// SIMATIC S7-200 project (STEP 7-Micro/WIN), CPU 226 CN REL 02.01

ORGANIZATION_BLOCK MAIN:OB1
TITLE=程序注释
BEGIN
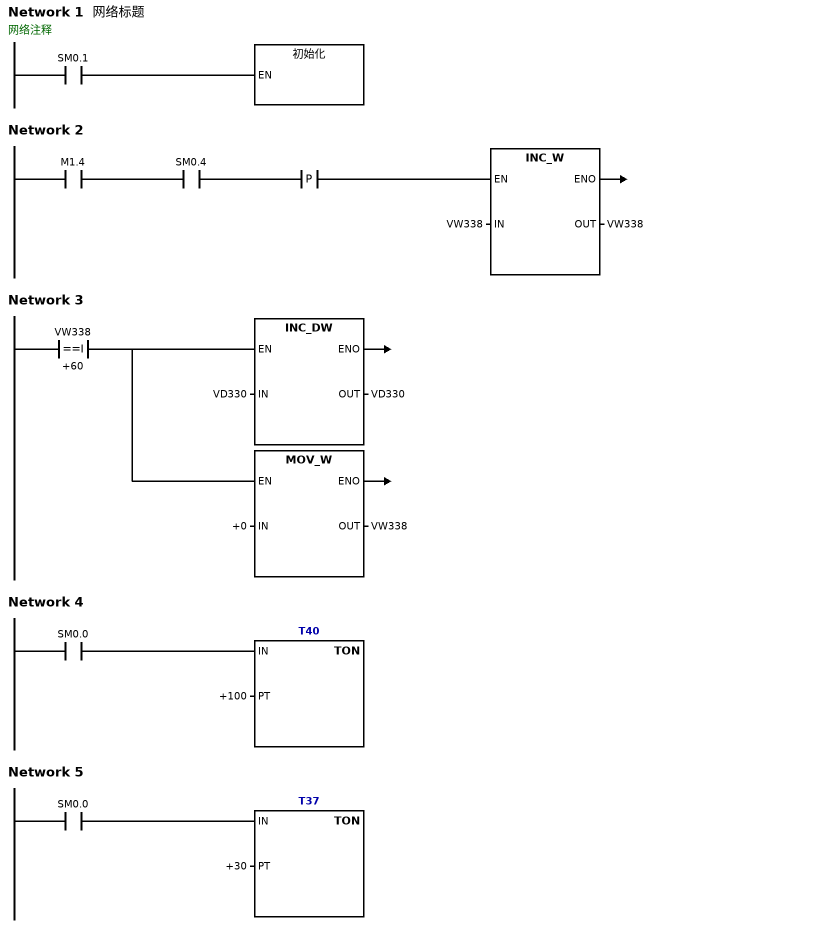
Network 1 // 网络标题
// 网络注释
LD     SM0.1
CALL   初始化:SBR0
Network 2
LD     M1.4
A      SM0.4
EU
INCW   VW338
Network 3
LDW=   VW338, +60
INCD   VD330
MOVW   +0, VW338
Network 4
LD     SM0.0
TON    T40, +100
Network 5
LD     SM0.0
TON    T37, +30
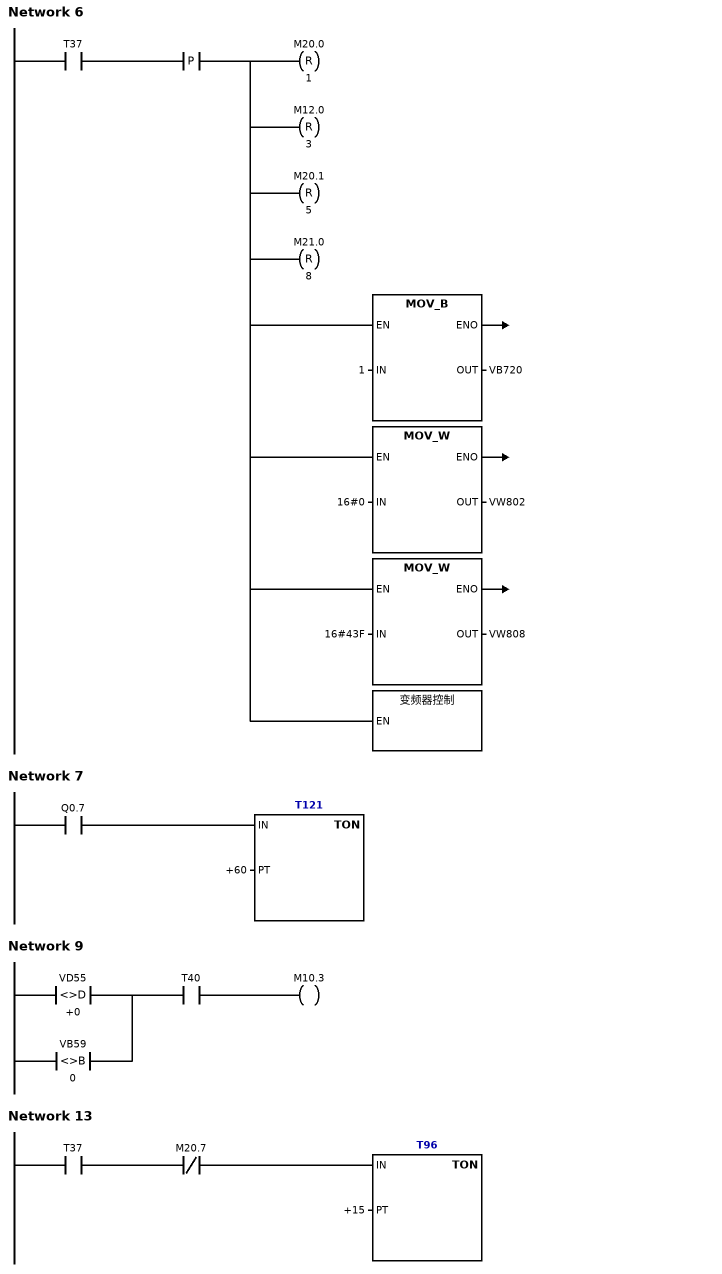
Network 6
LD     T37
EU
R      M20.0, 1
R      M12.0, 3
R      M20.1, 5
R      M21.0, 8
MOVB   1, VB720
MOVW   16#0, VW802
MOVW   16#43F, VW808
CALL   变频器控制:SBR16
Network 7
LD     Q0.7
TON    T121, +60
Network 9
LDD<>  VD55, +0
OB<>   VB59, 0
A      T40
=      M10.3
Network 13
LD     T37
AN     M20.7
TON    T96, +15
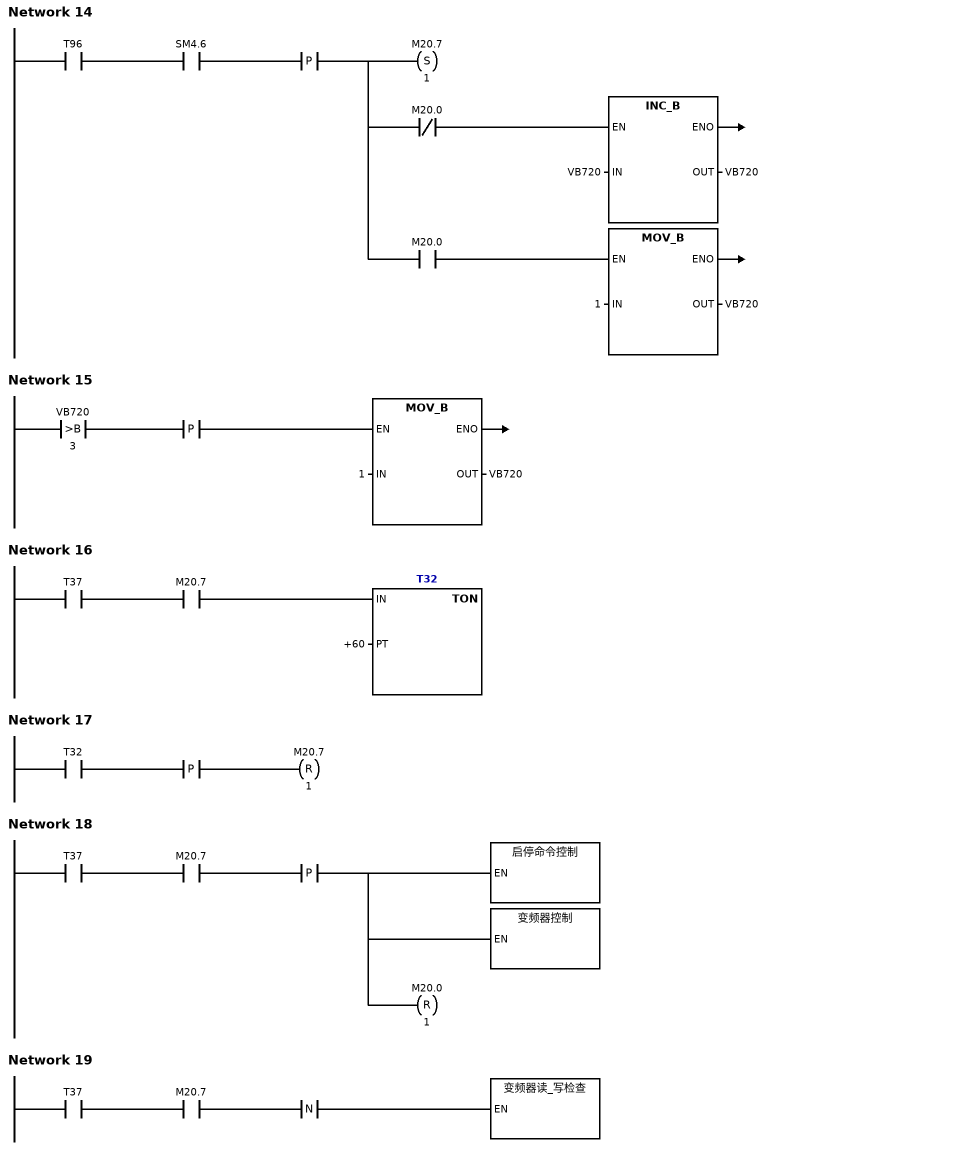
Network 14
LD     T96
A      SM4.6
EU
LPS
S      M20.7, 1
AN     M20.0
INCB   VB720
LPP
A      M20.0
MOVB   1, VB720
Network 15
LDB>   VB720, 3
EU
MOVB   1, VB720
Network 16
LD     T37
A      M20.7
TON    T32, +60
Network 17
LD     T32
EU
R      M20.7, 1
Network 18
LD     T37
A      M20.7
EU
CALL   启停命令控制:SBR4
CALL   变频器控制:SBR16
R      M20.0, 1
Network 19
LD     T37
A      M20.7
ED
CALL   变频器读_写检查:SBR3
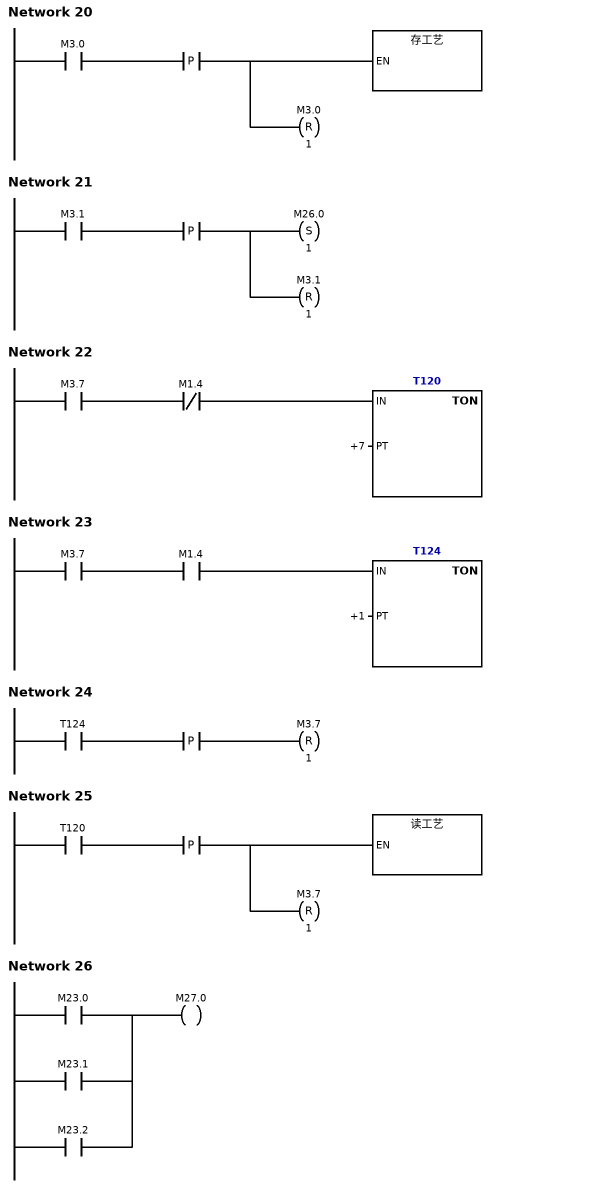
Network 20
LD     M3.0
EU
CALL   存工艺:SBR5
R      M3.0, 1
Network 21
LD     M3.1
EU
S      M26.0, 1
R      M3.1, 1
Network 22
LD     M3.7
AN     M1.4
TON    T120, +7
Network 23
LD     M3.7
A      M1.4
TON    T124, +1
Network 24
LD     T124
EU
R      M3.7, 1
Network 25
LD     T120
EU
CALL   读工艺:SBR6
R      M3.7, 1
Network 26
LD     M23.0
O      M23.1
O      M23.2
=      M27.0
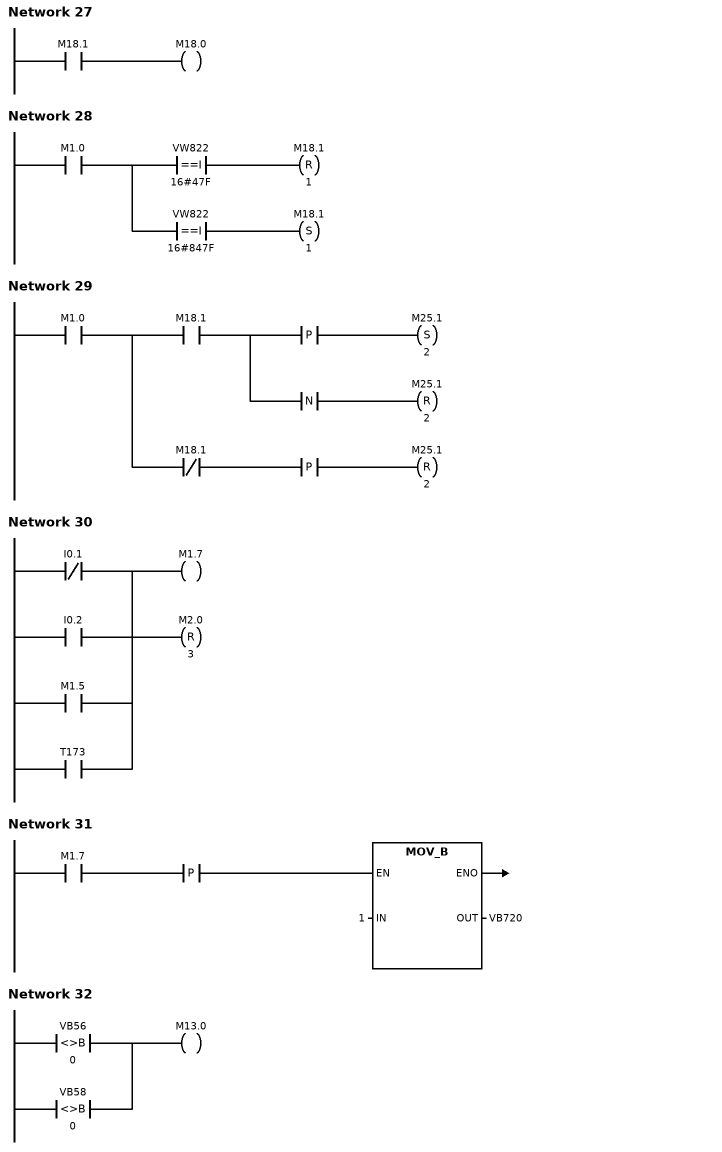
Network 27
LD     M18.1
=      M18.0
Network 28
LD     M1.0
LPS
AW=    VW822, 16#47F
R      M18.1, 1
LPP
AW=    VW822, 16#847F
S      M18.1, 1
Network 29
LD     M1.0
LPS
A      M18.1
LPS
EU
S      M25.1, 2
LPP
ED
R      M25.1, 2
LPP
AN     M18.1
EU
R      M25.1, 2
Network 30
LDN    I0.1
O      I0.2
O      M1.5
O      T173
=      M1.7
R      M2.0, 3
Network 31
LD     M1.7
EU
MOVB   1, VB720
Network 32
LDB<>  VB56, 0
OB<>   VB58, 0
=      M13.0
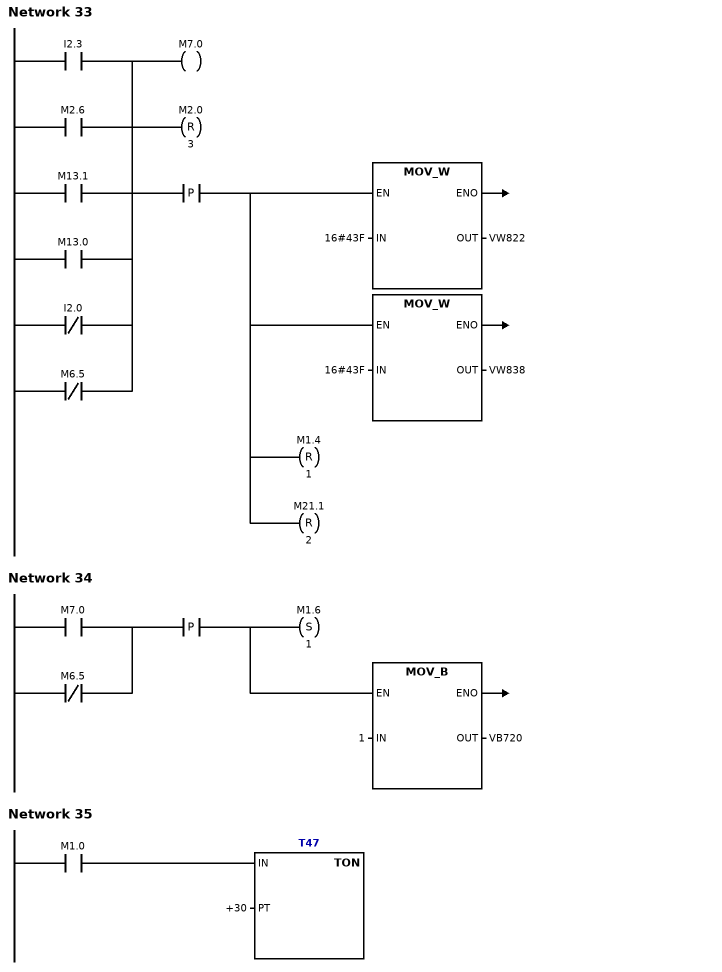
Network 33
LD     I2.3
O      M2.6
O      M13.1
O      M13.0
ON     I2.0
ON     M6.5
=      M7.0
R      M2.0, 3
EU
MOVW   16#43F, VW822
MOVW   16#43F, VW838
R      M1.4, 1
R      M21.1, 2
Network 34
LD     M7.0
ON     M6.5
EU
S      M1.6, 1
MOVB   1, VB720
Network 35
LD     M1.0
TON    T47, +30
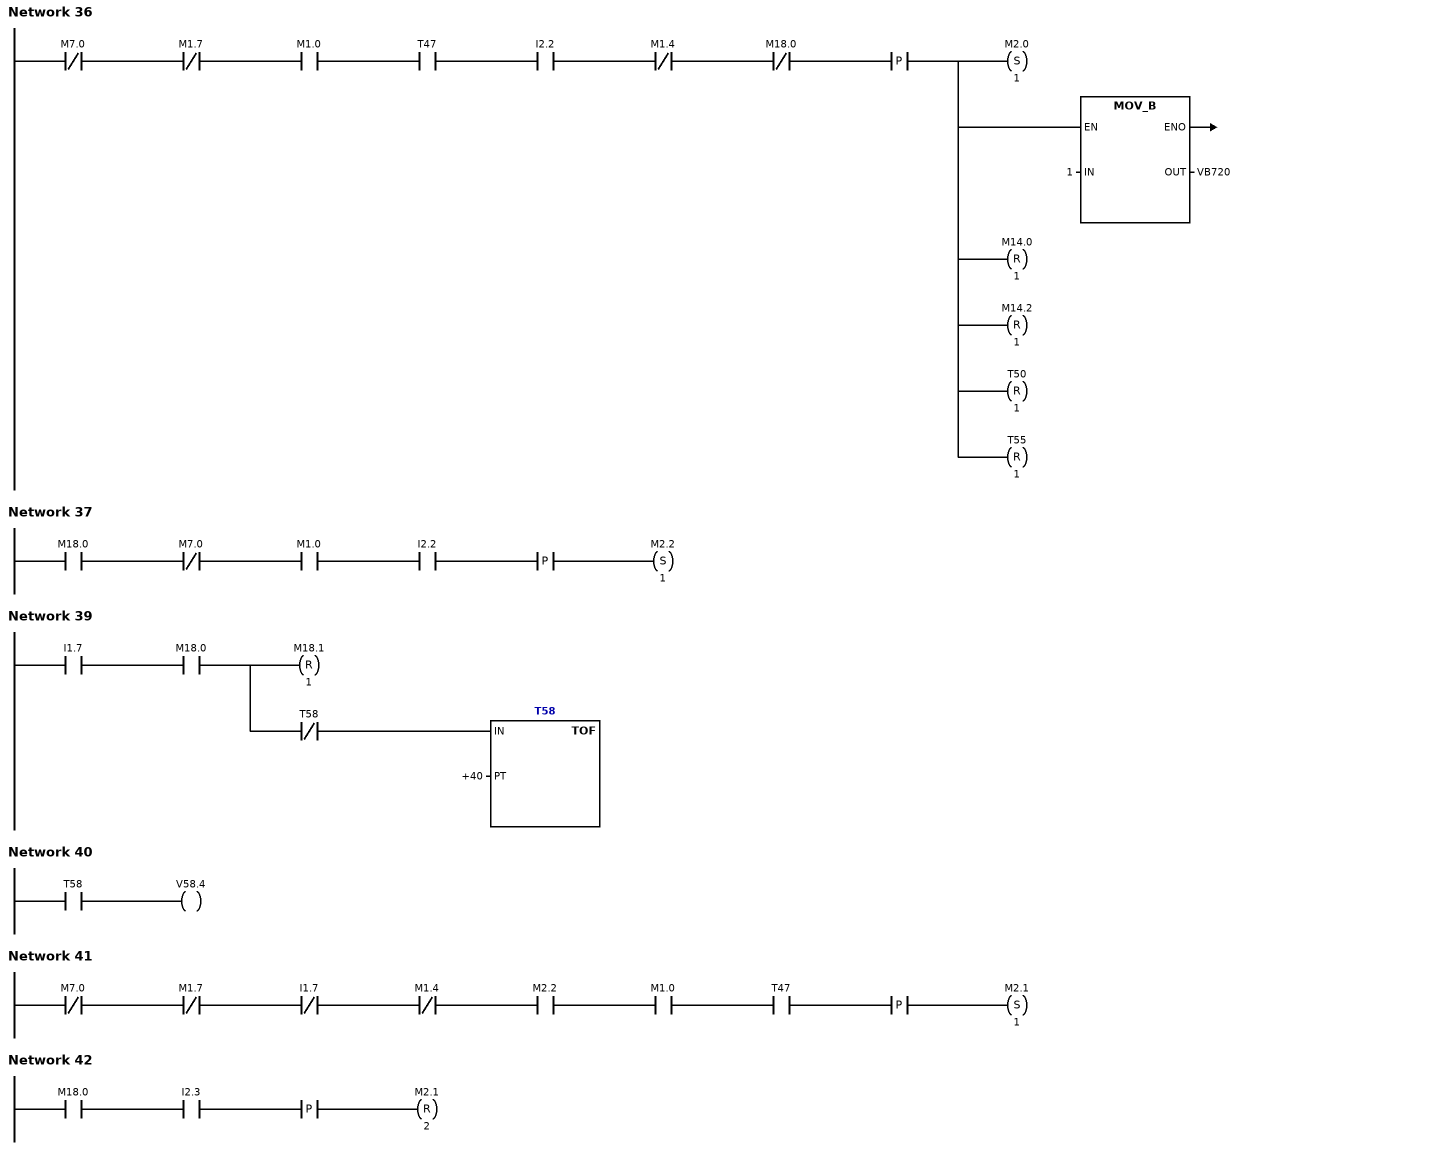
Network 36
LDN    M7.0
AN     M1.7
A      M1.0
A      T47
A      I2.2
AN     M1.4
AN     M18.0
EU
S      M2.0, 1
MOVB   1, VB720
R      M14.0, 1
R      M14.2, 1
R      T50, 1
R      T55, 1
Network 37
LD     M18.0
AN     M7.0
A      M1.0
A      I2.2
EU
S      M2.2, 1
Network 39
LD     I1.7
A      M18.0
R      M18.1, 1
AN     T58
TOF    T58, +40
Network 40
LD     T58
=      V58.4
Network 41
LDN    M7.0
AN     M1.7
AN     I1.7
AN     M1.4
A      M2.2
A      M1.0
A      T47
EU
S      M2.1, 1
Network 42
LD     M18.0
A      I2.3
EU
R      M2.1, 2
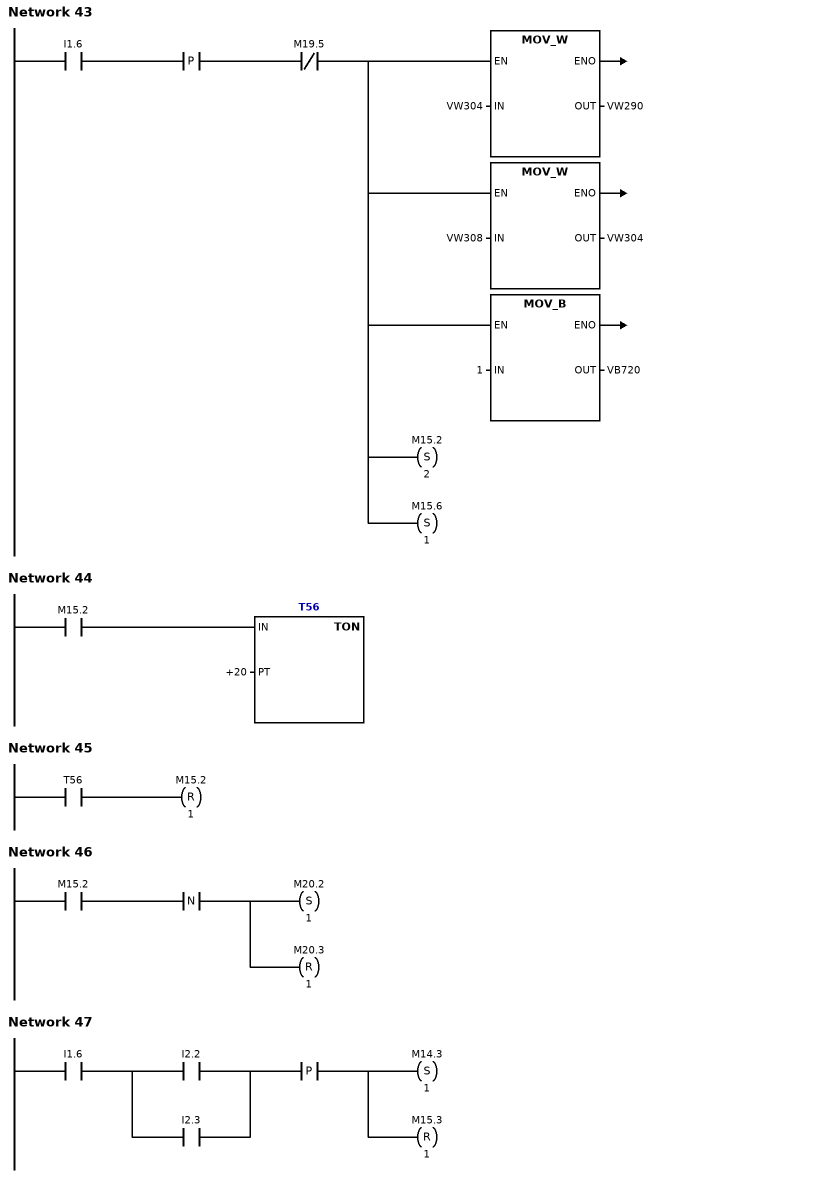
Network 43
LD     I1.6
EU
AN     M19.5
MOVW   VW304, VW290
MOVW   VW308, VW304
MOVB   1, VB720
S      M15.2, 2
S      M15.6, 1
Network 44
LD     M15.2
TON    T56, +20
Network 45
LD     T56
R      M15.2, 1
Network 46
LD     M15.2
ED
S      M20.2, 1
R      M20.3, 1
Network 47
LD     I1.6
LD     I2.2
O      I2.3
ALD
EU
S      M14.3, 1
R      M15.3, 1
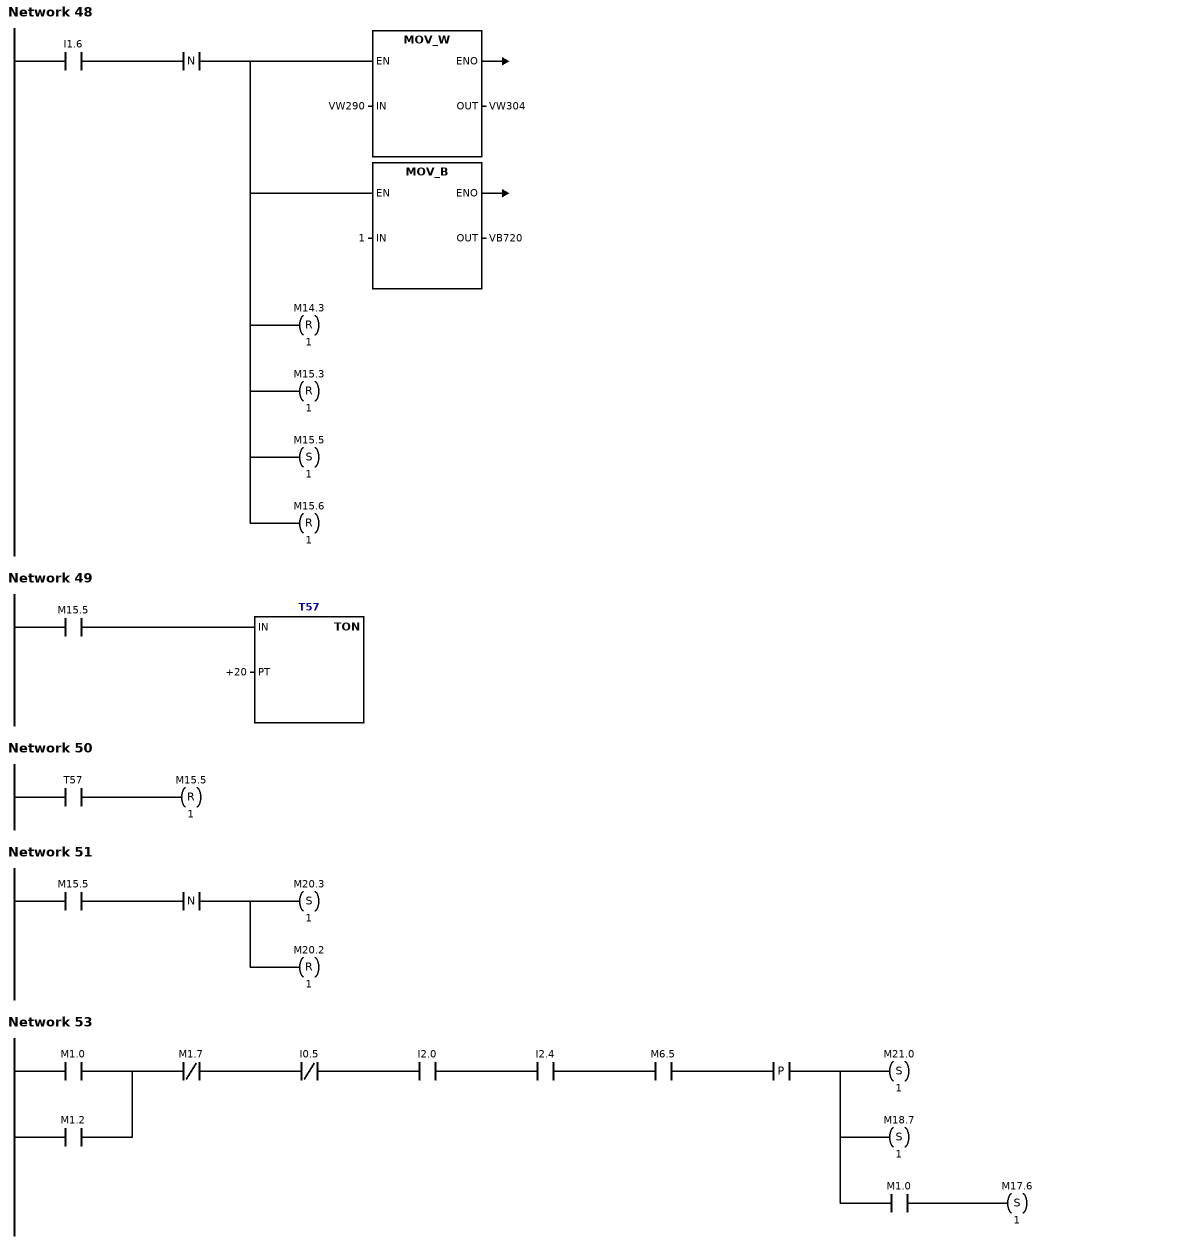
Network 48
LD     I1.6
ED
MOVW   VW290, VW304
MOVB   1, VB720
R      M14.3, 1
R      M15.3, 1
S      M15.5, 1
R      M15.6, 1
Network 49
LD     M15.5
TON    T57, +20
Network 50
LD     T57
R      M15.5, 1
Network 51
LD     M15.5
ED
S      M20.3, 1
R      M20.2, 1
Network 53
LD     M1.0
O      M1.2
AN     M1.7
AN     I0.5
A      I2.0
A      I2.4
A      M6.5
EU
S      M21.0, 1
S      M18.7, 1
A      M1.0
S      M17.6, 1
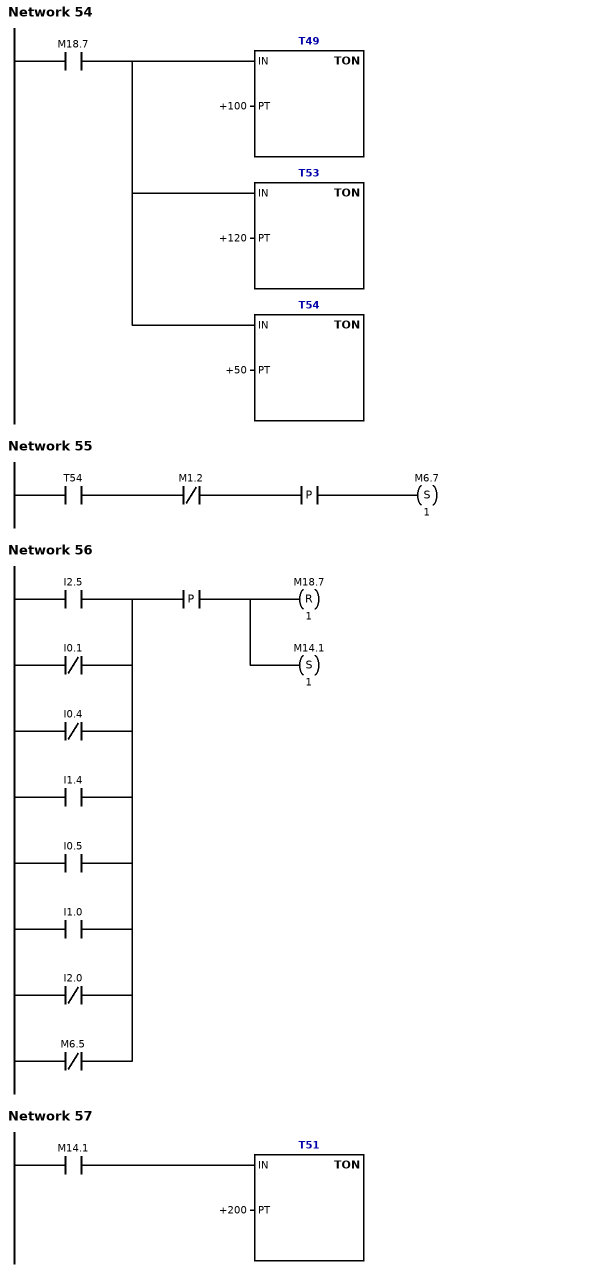
Network 54
LD     M18.7
TON    T49, +100
TON    T53, +120
TON    T54, +50
Network 55
LD     T54
AN     M1.2
EU
S      M6.7, 1
Network 56
LD     I2.5
ON     I0.1
ON     I0.4
O      I1.4
O      I0.5
O      I1.0
ON     I2.0
ON     M6.5
EU
R      M18.7, 1
S      M14.1, 1
Network 57
LD     M14.1
TON    T51, +200
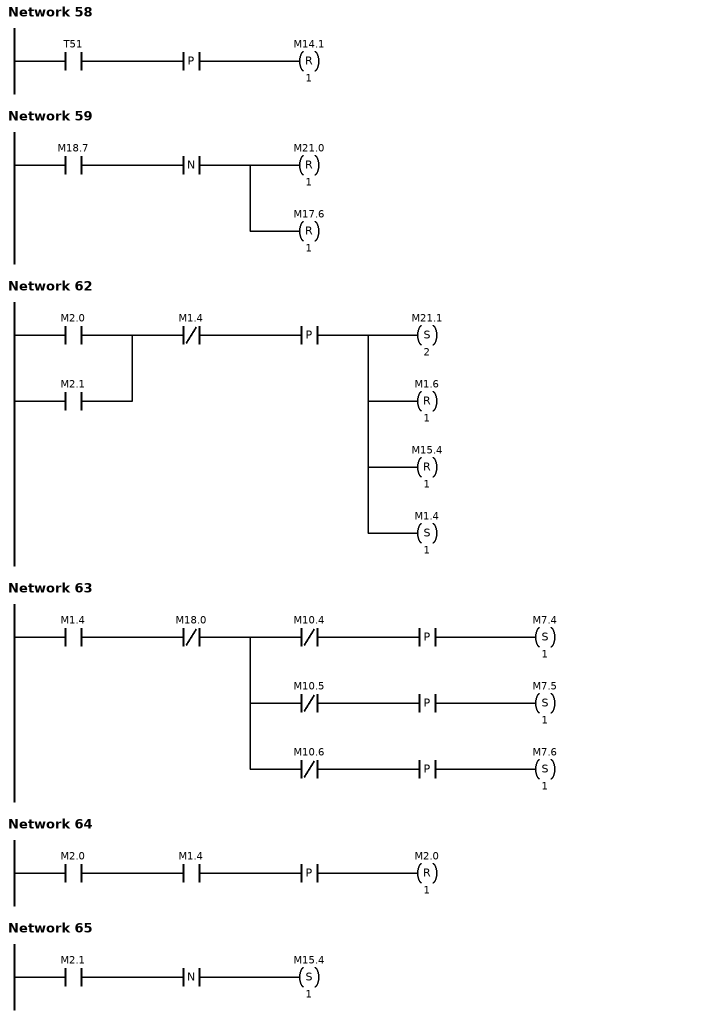
Network 58
LD     T51
EU
R      M14.1, 1
Network 59
LD     M18.7
ED
R      M21.0, 1
R      M17.6, 1
Network 62
LD     M2.0
O      M2.1
AN     M1.4
EU
S      M21.1, 2
R      M1.6, 1
R      M15.4, 1
S      M1.4, 1
Network 63
LD     M1.4
AN     M18.0
LPS
AN     M10.4
EU
S      M7.4, 1
LRD
AN     M10.5
EU
S      M7.5, 1
LPP
AN     M10.6
EU
S      M7.6, 1
Network 64
LD     M2.0
A      M1.4
EU
R      M2.0, 1
Network 65
LD     M2.1
ED
S      M15.4, 1
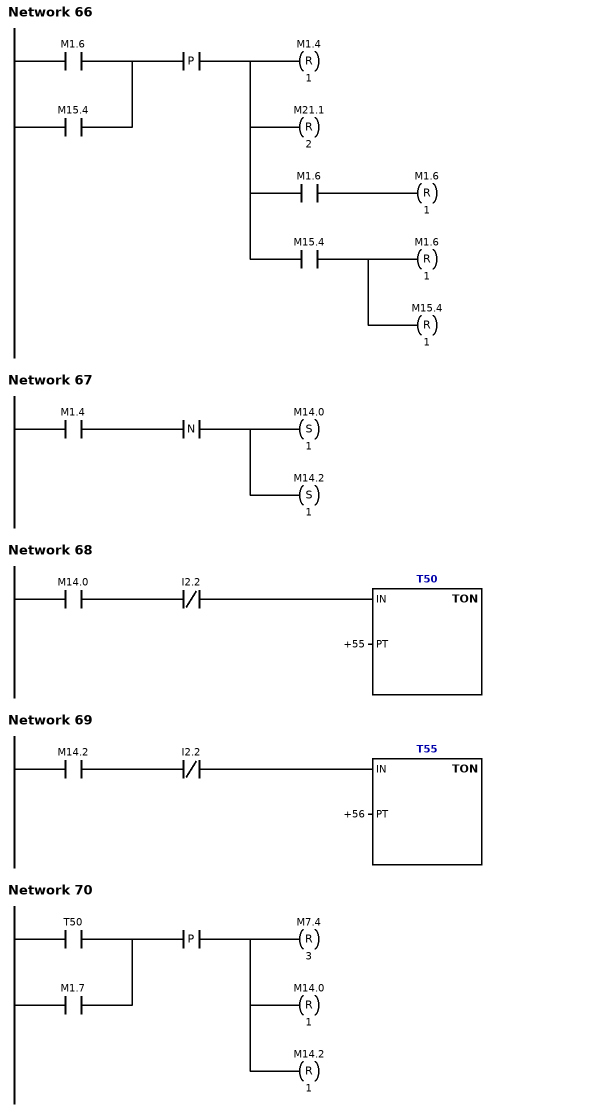
Network 66
LD     M1.6
O      M15.4
EU
LPS
R      M1.4, 1
R      M21.1, 2
A      M1.6
R      M1.6, 1
LPP
A      M15.4
R      M1.6, 1
R      M15.4, 1
Network 67
LD     M1.4
ED
S      M14.0, 1
S      M14.2, 1
Network 68
LD     M14.0
AN     I2.2
TON    T50, +55
Network 69
LD     M14.2
AN     I2.2
TON    T55, +56
Network 70
LD     T50
O      M1.7
EU
R      M7.4, 3
R      M14.0, 1
R      M14.2, 1
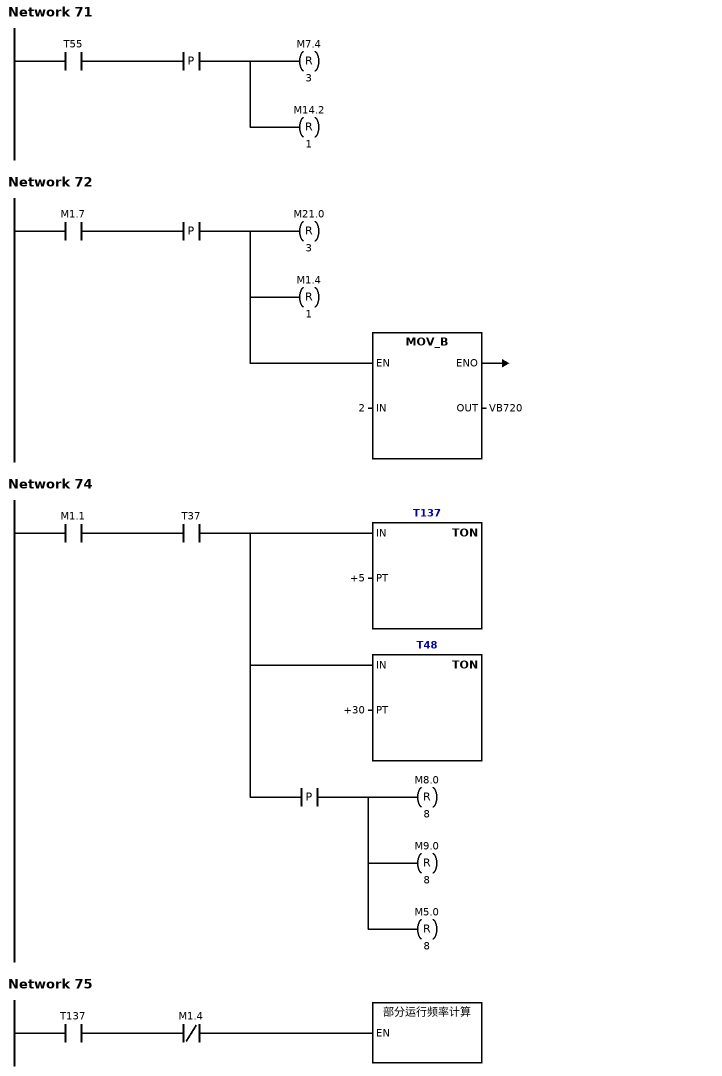
Network 71
LD     T55
EU
R      M7.4, 3
R      M14.2, 1
Network 72
LD     M1.7
EU
R      M21.0, 3
R      M1.4, 1
MOVB   2, VB720
Network 74
LD     M1.1
A      T37
TON    T137, +5
TON    T48, +30
EU
R      M8.0, 8
R      M9.0, 8
R      M5.0, 8
Network 75
LD     T137
AN     M1.4
CALL   部分运行频率计算:SBR11
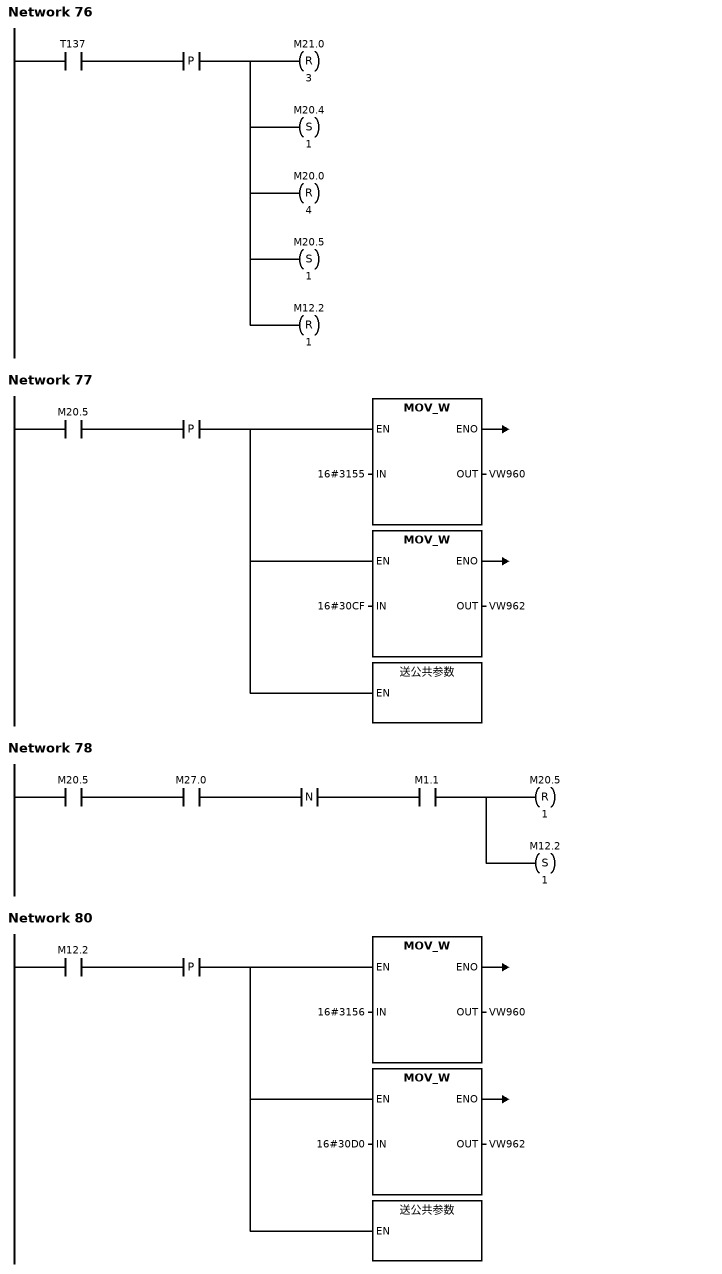
Network 76
LD     T137
EU
R      M21.0, 3
S      M20.4, 1
R      M20.0, 4
S      M20.5, 1
R      M12.2, 1
Network 77
LD     M20.5
EU
MOVW   16#3155, VW960
MOVW   16#30CF, VW962
CALL   送公共参数:SBR13
Network 78
LD     M20.5
A      M27.0
ED
A      M1.1
R      M20.5, 1
S      M12.2, 1
Network 80
LD     M12.2
EU
MOVW   16#3156, VW960
MOVW   16#30D0, VW962
CALL   送公共参数:SBR13
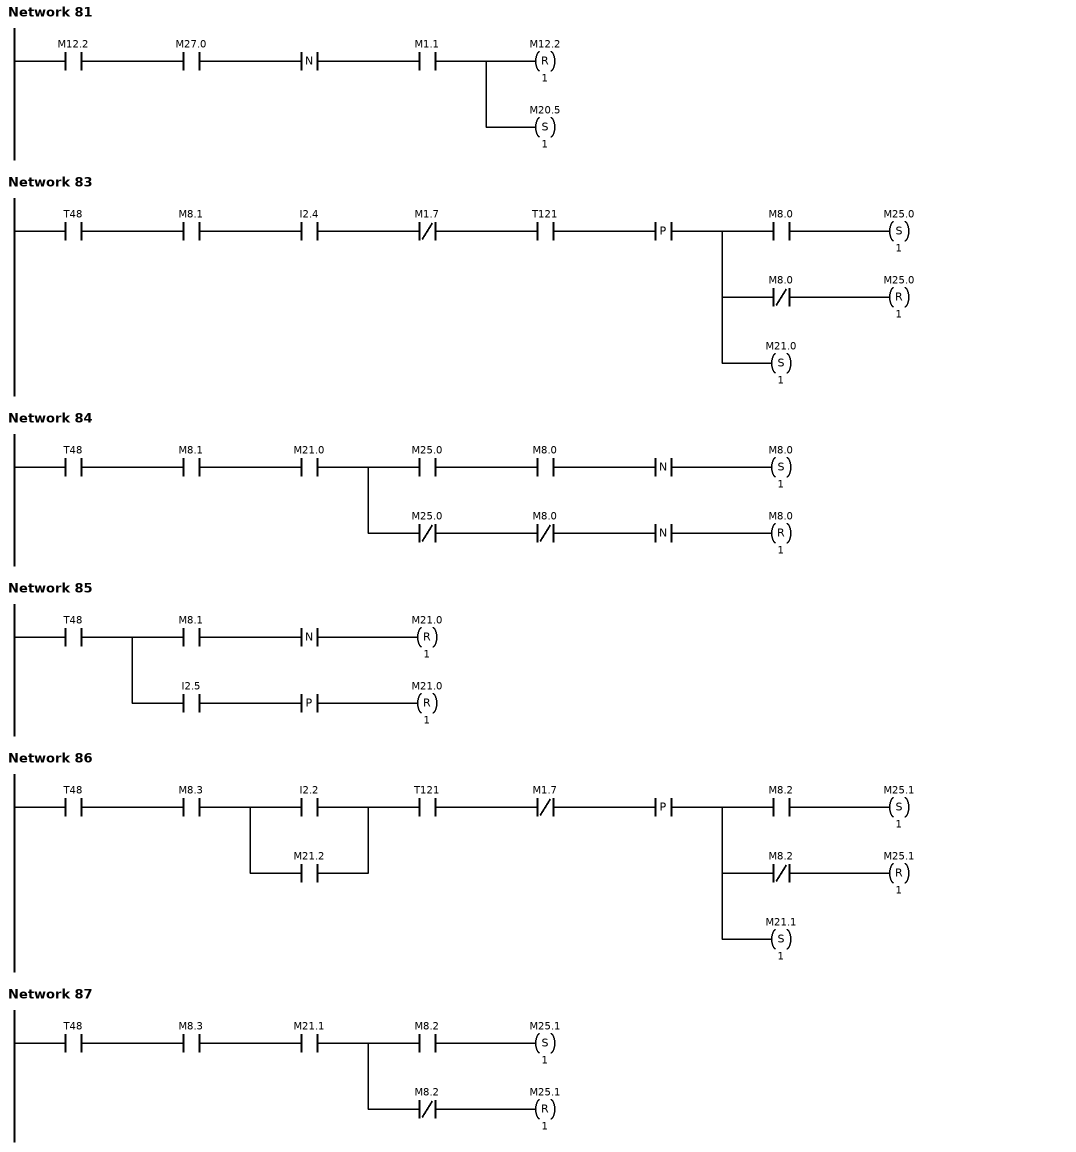
Network 81
LD     M12.2
A      M27.0
ED
A      M1.1
R      M12.2, 1
S      M20.5, 1
Network 83
LD     T48
A      M8.1
A      I2.4
AN     M1.7
A      T121
EU
LPS
A      M8.0
S      M25.0, 1
LRD
AN     M8.0
R      M25.0, 1
LPP
S      M21.0, 1
Network 84
LD     T48
A      M8.1
A      M21.0
LPS
A      M25.0
A      M8.0
ED
S      M8.0, 1
LPP
AN     M25.0
AN     M8.0
ED
R      M8.0, 1
Network 85
LD     T48
LPS
A      M8.1
ED
R      M21.0, 1
LPP
A      I2.5
EU
R      M21.0, 1
Network 86
LD     T48
A      M8.3
LD     I2.2
O      M21.2
ALD
A      T121
AN     M1.7
EU
LPS
A      M8.2
S      M25.1, 1
LRD
AN     M8.2
R      M25.1, 1
LPP
S      M21.1, 1
Network 87
LD     T48
A      M8.3
A      M21.1
LPS
A      M8.2
S      M25.1, 1
LPP
AN     M8.2
R      M25.1, 1
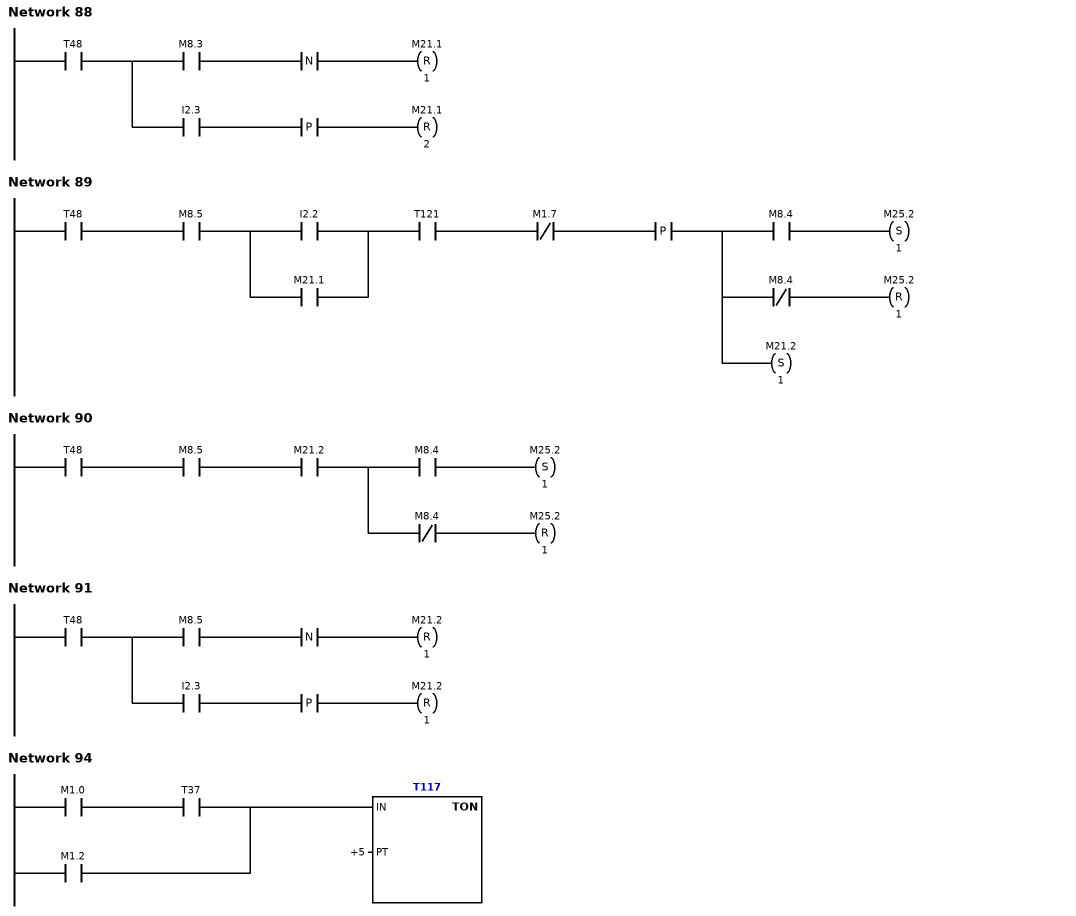
Network 88
LD     T48
LPS
A      M8.3
ED
R      M21.1, 1
LPP
A      I2.3
EU
R      M21.1, 2
Network 89
LD     T48
A      M8.5
LD     I2.2
O      M21.1
ALD
A      T121
AN     M1.7
EU
LPS
A      M8.4
S      M25.2, 1
LRD
AN     M8.4
R      M25.2, 1
LPP
S      M21.2, 1
Network 90
LD     T48
A      M8.5
A      M21.2
LPS
A      M8.4
S      M25.2, 1
LPP
AN     M8.4
R      M25.2, 1
Network 91
LD     T48
LPS
A      M8.5
ED
R      M21.2, 1
LPP
A      I2.3
EU
R      M21.2, 1
Network 94
LD     M1.0
A      T37
O      M1.2
TON    T117, +5
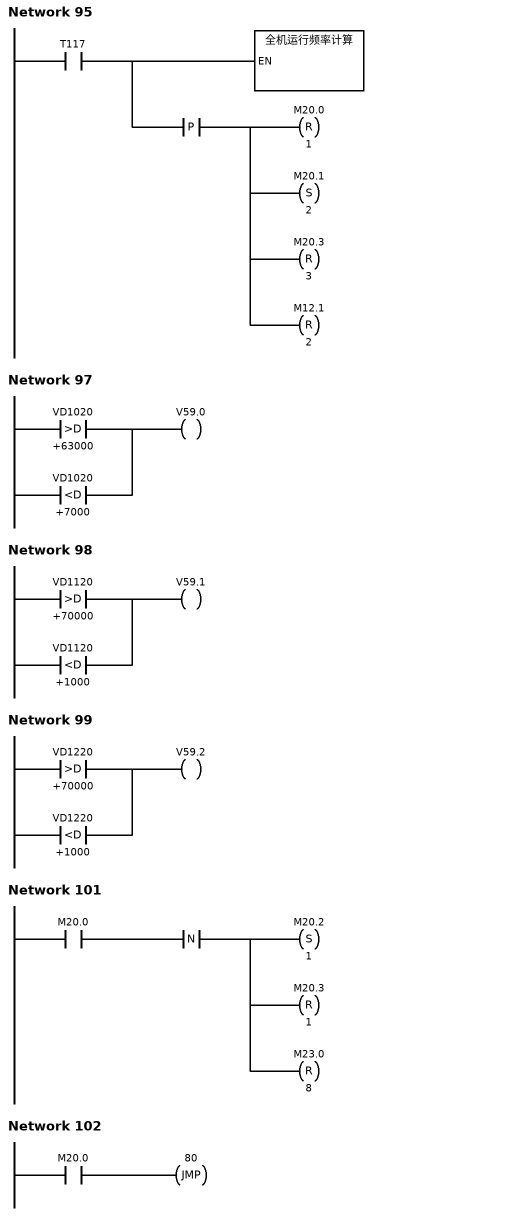
Network 95
LD     T117
CALL   全机运行频率计算:SBR10
EU
R      M20.0, 1
S      M20.1, 2
R      M20.3, 3
R      M12.1, 2
Network 97
LDD>   VD1020, +63000
OD<    VD1020, +7000
=      V59.0
Network 98
LDD>   VD1120, +70000
OD<    VD1120, +1000
=      V59.1
Network 99
LDD>   VD1220, +70000
OD<    VD1220, +1000
=      V59.2
Network 101
LD     M20.0
ED
S      M20.2, 1
R      M20.3, 1
R      M23.0, 8
Network 102
LD     M20.0
JMP    80
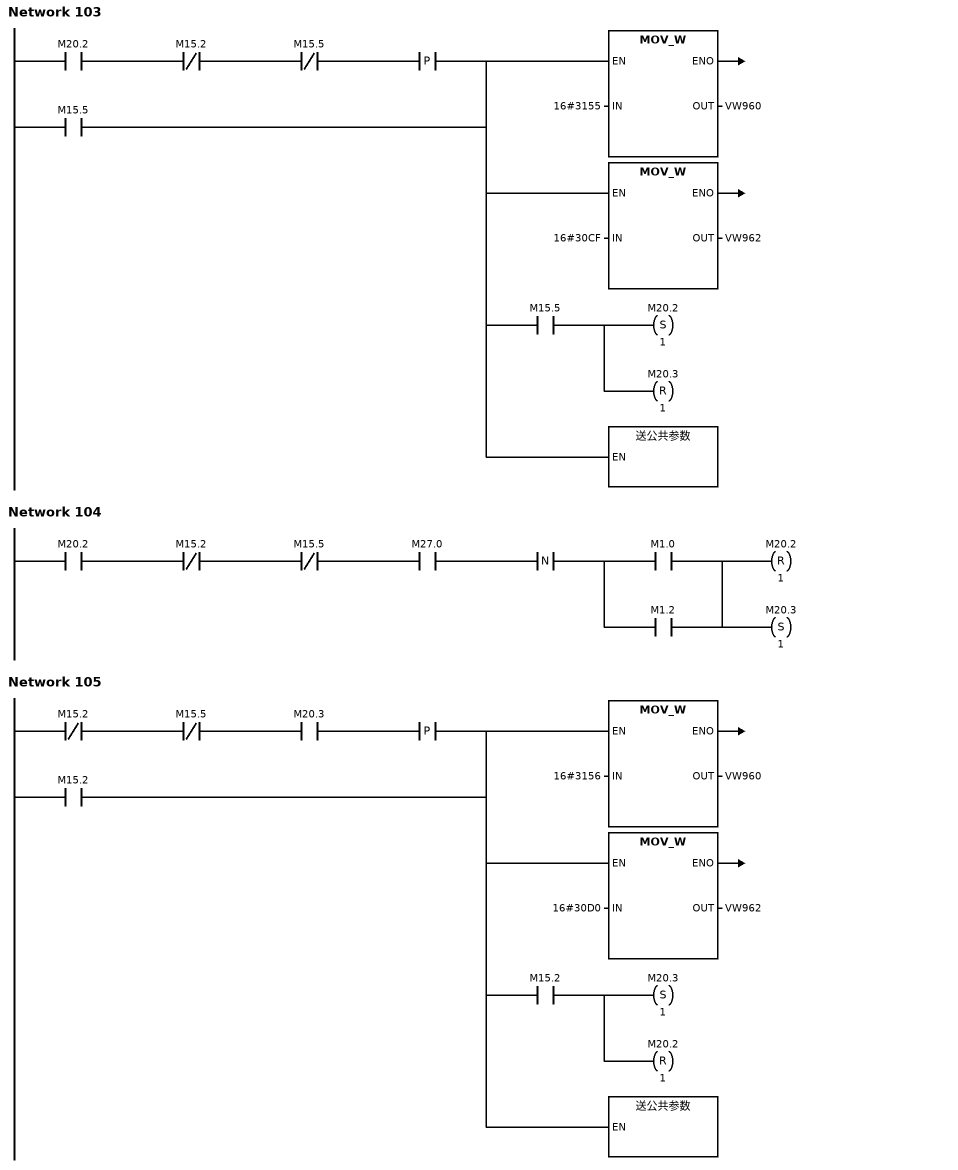
Network 103
LD     M20.2
AN     M15.2
AN     M15.5
EU
O      M15.5
LPS
MOVW   16#3155, VW960
MOVW   16#30CF, VW962
A      M15.5
S      M20.2, 1
R      M20.3, 1
LPP
CALL   送公共参数:SBR13
Network 104
LD     M20.2
AN     M15.2
AN     M15.5
A      M27.0
ED
LD     M1.0
O      M1.2
ALD
R      M20.2, 1
S      M20.3, 1
Network 105
LDN    M15.2
AN     M15.5
A      M20.3
EU
O      M15.2
LPS
MOVW   16#3156, VW960
MOVW   16#30D0, VW962
A      M15.2
S      M20.3, 1
R      M20.2, 1
LPP
CALL   送公共参数:SBR13
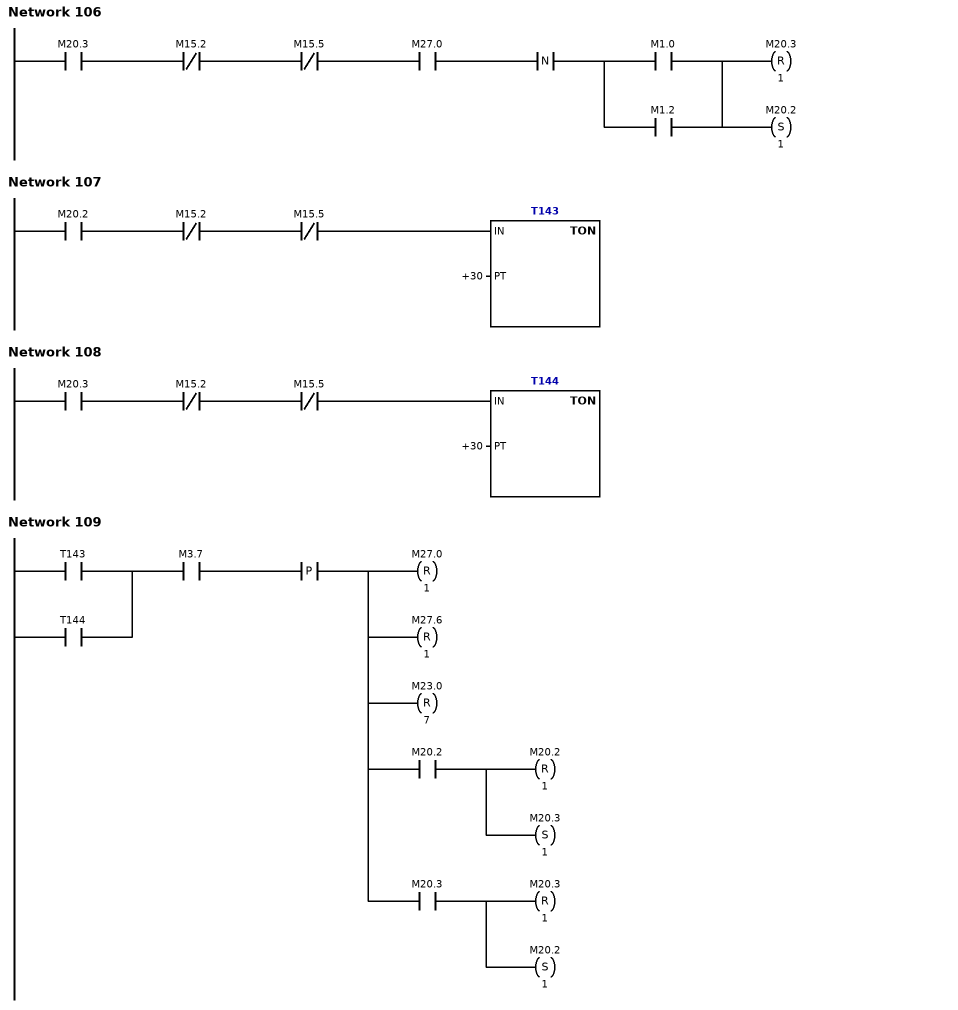
Network 106
LD     M20.3
AN     M15.2
AN     M15.5
A      M27.0
ED
LD     M1.0
O      M1.2
ALD
R      M20.3, 1
S      M20.2, 1
Network 107
LD     M20.2
AN     M15.2
AN     M15.5
TON    T143, +30
Network 108
LD     M20.3
AN     M15.2
AN     M15.5
TON    T144, +30
Network 109
LD     T143
O      T144
A      M3.7
EU
LPS
R      M27.0, 1
R      M27.6, 1
R      M23.0, 7
A      M20.2
R      M20.2, 1
S      M20.3, 1
LPP
A      M20.3
R      M20.3, 1
S      M20.2, 1
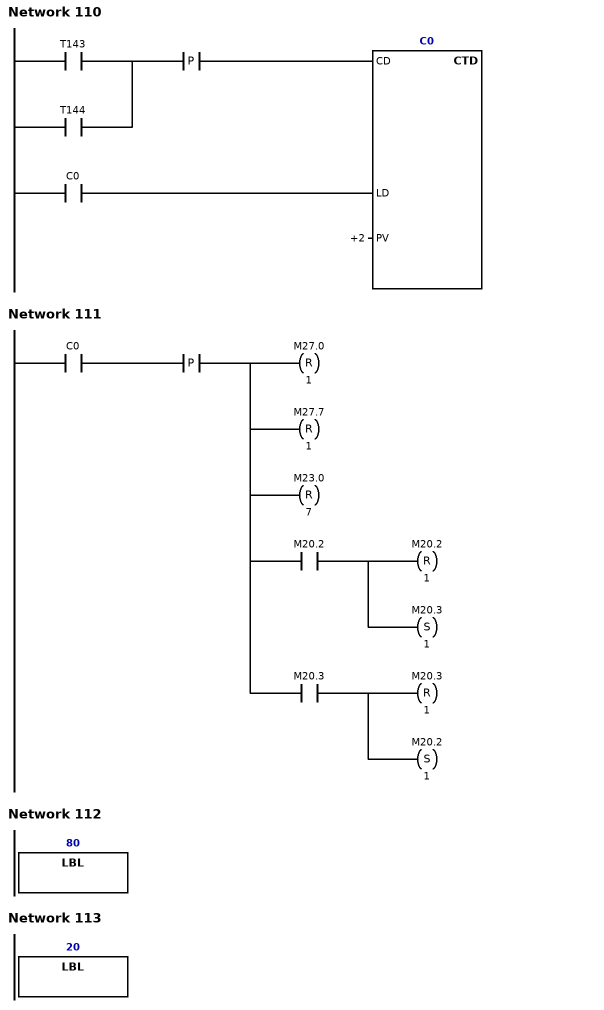
Network 110
LD     T143
O      T144
EU
LD     C0
CTD    C0, +2
Network 111
LD     C0
EU
LPS
R      M27.0, 1
R      M27.7, 1
R      M23.0, 7
A      M20.2
R      M20.2, 1
S      M20.3, 1
LPP
A      M20.3
R      M20.3, 1
S      M20.2, 1
Network 112
LBL    80
Network 113
LBL    20
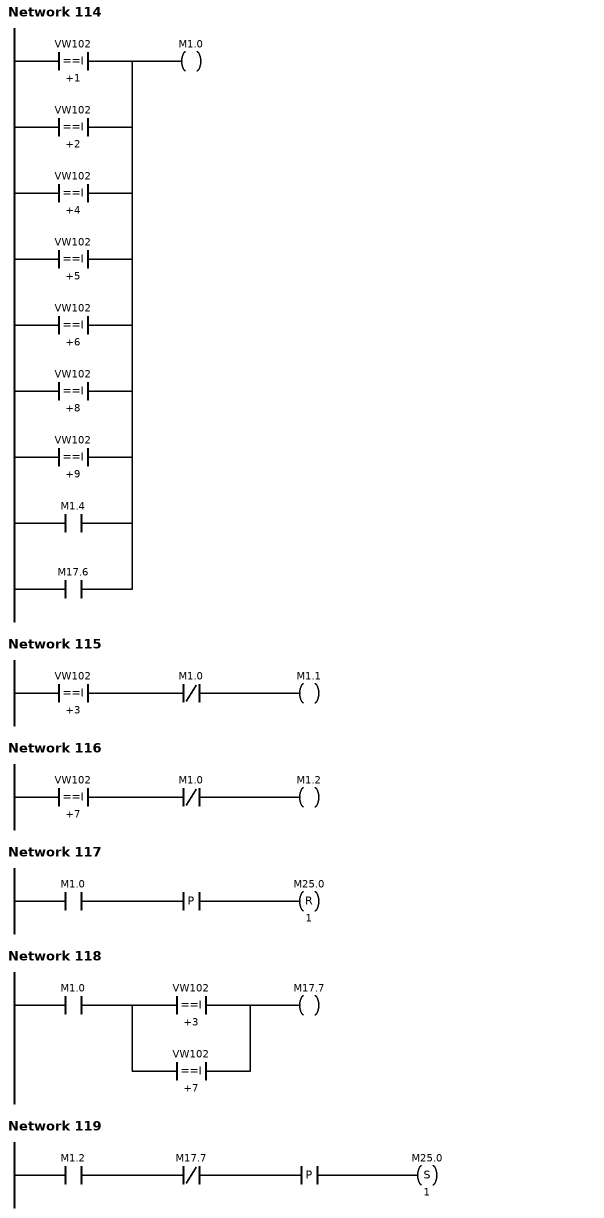
Network 114
LDW=   VW102, +1
OW=    VW102, +2
OW=    VW102, +4
OW=    VW102, +5
OW=    VW102, +6
OW=    VW102, +8
OW=    VW102, +9
O      M1.4
O      M17.6
=      M1.0
Network 115
LDW=   VW102, +3
AN     M1.0
=      M1.1
Network 116
LDW=   VW102, +7
AN     M1.0
=      M1.2
Network 117
LD     M1.0
EU
R      M25.0, 1
Network 118
LD     M1.0
LDW=   VW102, +3
OW=    VW102, +7
ALD
=      M17.7
Network 119
LD     M1.2
AN     M17.7
EU
S      M25.0, 1
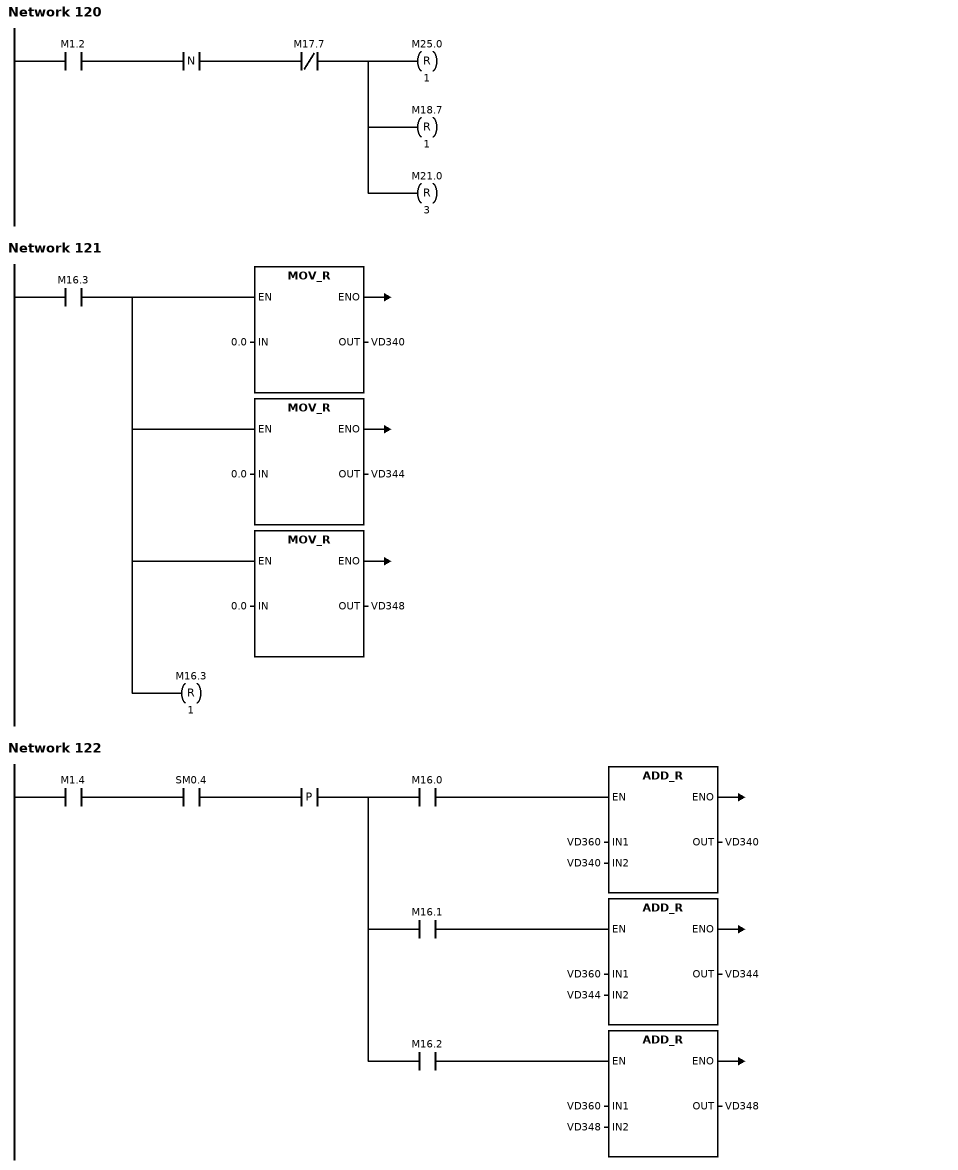
Network 120
LD     M1.2
ED
AN     M17.7
R      M25.0, 1
R      M18.7, 1
R      M21.0, 3
Network 121
LD     M16.3
MOVR   0.0, VD340
MOVR   0.0, VD344
MOVR   0.0, VD348
R      M16.3, 1
Network 122
LD     M1.4
A      SM0.4
EU
LPS
A      M16.0
+R     VD360, VD340
LRD
A      M16.1
+R     VD360, VD344
LPP
A      M16.2
+R     VD360, VD348
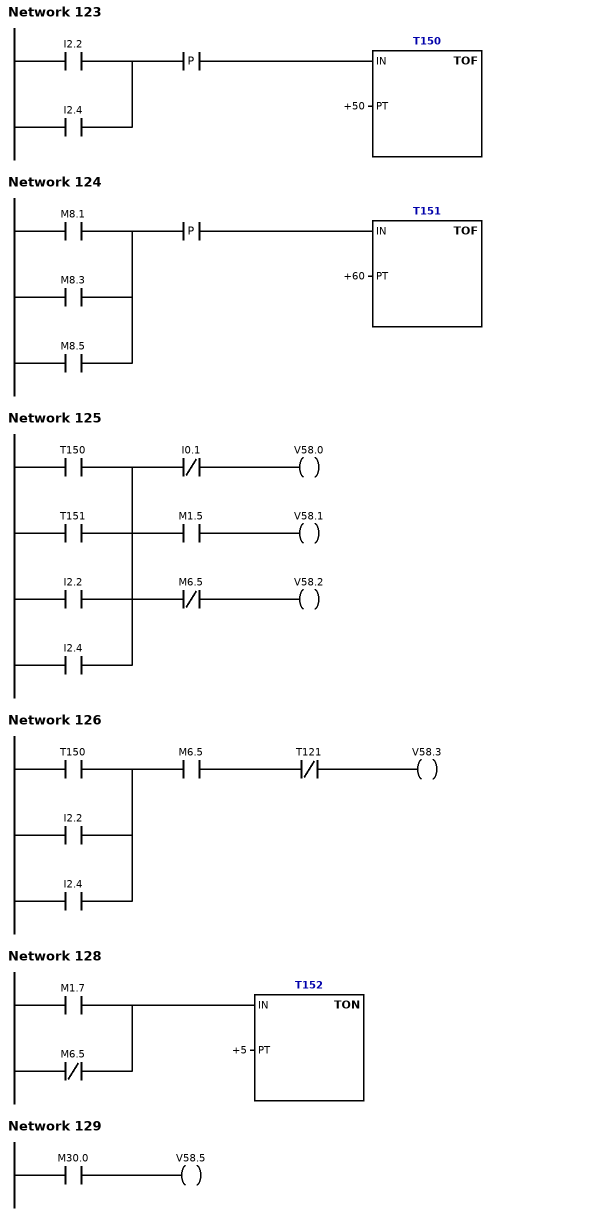
Network 123
LD     I2.2
O      I2.4
EU
TOF    T150, +50
Network 124
LD     M8.1
O      M8.3
O      M8.5
EU
TOF    T151, +60
Network 125
LD     T150
O      T151
O      I2.2
O      I2.4
LPS
AN     I0.1
=      V58.0
LRD
A      M1.5
=      V58.1
LPP
AN     M6.5
=      V58.2
Network 126
LD     T150
O      I2.2
O      I2.4
A      M6.5
AN     T121
=      V58.3
Network 128
LD     M1.7
ON     M6.5
TON    T152, +5
Network 129
LD     M30.0
=      V58.5
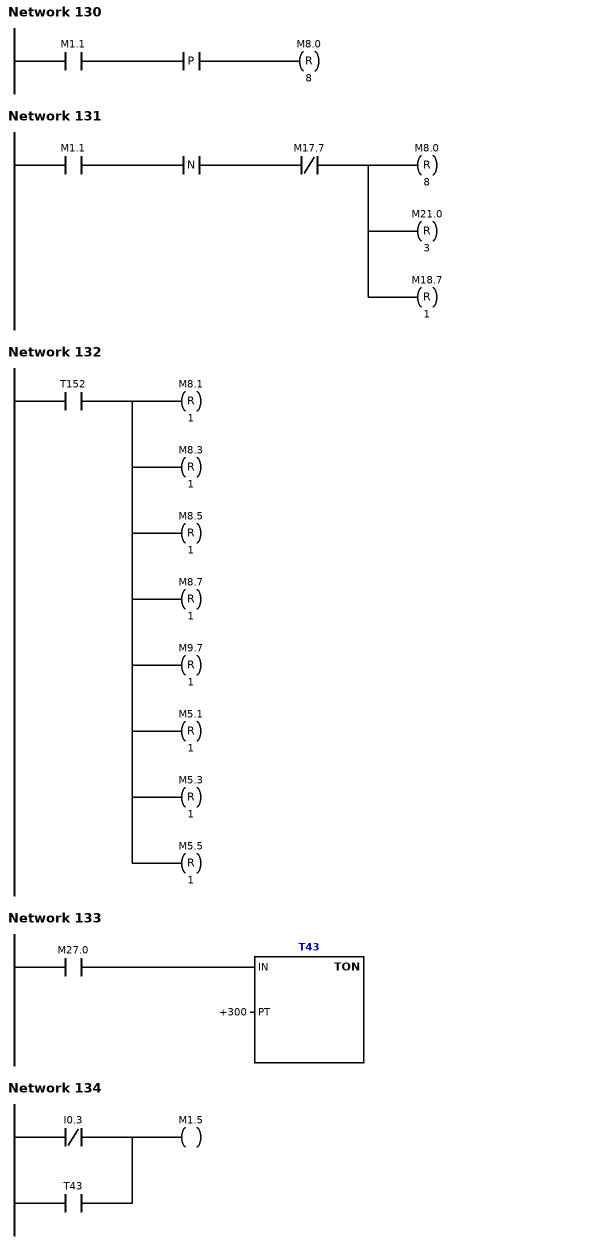
Network 130
LD     M1.1
EU
R      M8.0, 8
Network 131
LD     M1.1
ED
AN     M17.7
R      M8.0, 8
R      M21.0, 3
R      M18.7, 1
Network 132
LD     T152
R      M8.1, 1
R      M8.3, 1
R      M8.5, 1
R      M8.7, 1
R      M9.7, 1
R      M5.1, 1
R      M5.3, 1
R      M5.5, 1
Network 133
LD     M27.0
TON    T43, +300
Network 134
LDN    I0.3
O      T43
=      M1.5
